// TIA Portal V17 export
// export: Created 2024-06-14T09:52:47.4803756Z, ExportSetting WithDefaults, DisplayName Totally Integrated Automation Portal, DisplayVersion V17, DisplayName TIA Portal Openness, DisplayVersion V17, DisplayName TIA Portal Version Control Interface, DisplayVersion V17, DisplayName Simotion SCOUT TIA, DisplayVersion 5.4.3.0, DisplayName SINAMICS Startdrive Advanced, DisplayVersion V17 SP1 Update 1, DisplayName SINAMICS Startdrive G110M, G120, G120C, G120D, G120P, G115D, DisplayVersion V17 SP1 Update 1, DisplayName SINAMICS Startdrive G130, G150, S120, S150, SINAMICS MV, S210, DisplayVersion V17 SP1 Update 1, DisplayName STEP 7 Professional, DisplayVersion V17, DisplayName STEP 7 Safety, DisplayVersion V17, DisplayName WinCC Professional, DisplayVersion V17
FUNCTION_BLOCK "FILLING_STATION4_FB"   // FB500, LAD
{ S7_Optimized_Access := 'TRUE' }
VERSION : 0.1
// stored: AutoNumber false, IsIECCheckEnabled false, IsRetainMemResEnabled false, MemoryReserve 100, SetENOAutomatically false, UDAEnableTagReadback false
   VAR
      STATION4_S1 { S7_SetPoint := 'True'} : "LPG_FILLING_FB";
      STATION4_S2 { S7_SetPoint := 'True'} : "LPG_FILLING_FB";
      STATION4_S3 { S7_SetPoint := 'True'} : "LPG_FILLING_FB";
      STATION4_S4 { S7_SetPoint := 'True'} : "LPG_FILLING_FB";
      STATION4_S5 { S7_SetPoint := 'True'} : "LPG_FILLING_FB";
      STATION4_S6 { S7_SetPoint := 'True'} : "LPG_FILLING_FB";
      FILLING_STATION4 { S7_SetPoint := 'True'} : "FILLING_FB";
      FILL_SEQ_STARTED { S7_SetPoint := 'True'} : Array[1..6] of Bool;
      FILLING_DONE : Array[1..6] of Bool;
   END_VAR
   VAR_TEMP   // added for the SCL form of the ladder/FBD networks
      _w1 : Bool;
   END_VAR
BEGIN

REGION Network 2: Call Filling Station-4
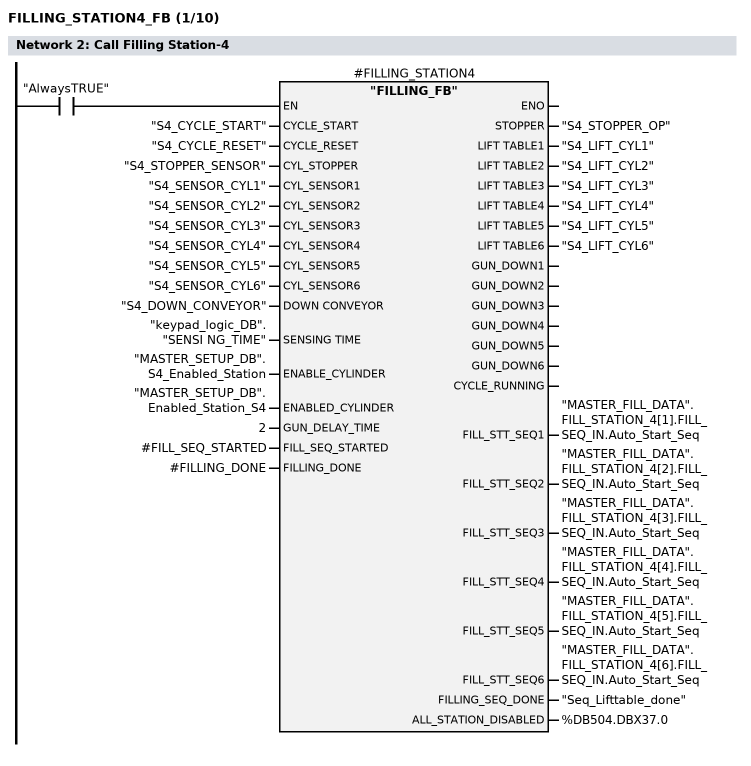
   RUNG wire#powerrail
      Contact( "AlwaysTRUE" )
      #FILLING_STATION4(CYCLE_START := "S4_CYCLE_START", CYCLE_RESET := "S4_CYCLE_RESET", CYL_STOPPER := "S4_STOPPER_SENSOR", CYL_SENSOR1 := "S4_SENSOR_CYL1", CYL_SENSOR2 := "S4_SENSOR_CYL2", CYL_SENSOR3 := "S4_SENSOR_CYL3", CYL_SENSOR4 := "S4_SENSOR_CYL4", CYL_SENSOR5 := "S4_SENSOR_CYL5", CYL_SENSOR6 := "S4_SENSOR_CYL6", "DOWN CONVEYOR" := "S4_DOWN_CONVEYOR", "SENSING TIME" := "keypad_logic_DB"."SENSI NG_TIME", ENABLE_CYLINDER := "MASTER_SETUP_DB".S4_Enabled_Station, ENABLED_CYLINDER := "MASTER_SETUP_DB".Enabled_Station_S4, GUN_DELAY_TIME := 2, FILL_SEQ_STARTED := #FILL_SEQ_STARTED, FILLING_DONE := #FILLING_DONE, STOPPER => "S4_STOPPER_OP", "LIFT TABLE1" => "S4_LIFT_CYL1", "LIFT TABLE2" => "S4_LIFT_CYL2", "LIFT TABLE3" => "S4_LIFT_CYL3", "LIFT TABLE4" => "S4_LIFT_CYL4", "LIFT TABLE5" => "S4_LIFT_CYL5", "LIFT TABLE6" => "S4_LIFT_CYL6", GUN_DOWN1 =>, GUN_DOWN2 =>, GUN_DOWN3 =>, GUN_DOWN4 =>, GUN_DOWN5 =>, GUN_DOWN6 =>, CYCLE_RUNNING =>, FILL_STT_SEQ1 => "MASTER_FILL_DATA".FILL_STATION_4[1].FILL_SEQ_IN.Auto_Start_Seq, FILL_STT_SEQ2 => "MASTER_FILL_DATA".FILL_STATION_4[2].FILL_SEQ_IN.Auto_Start_Seq, FILL_STT_SEQ3 => "MASTER_FILL_DATA".FILL_STATION_4[3].FILL_SEQ_IN.Auto_Start_Seq, FILL_STT_SEQ4 => "MASTER_FILL_DATA".FILL_STATION_4[4].FILL_SEQ_IN.Auto_Start_Seq, FILL_STT_SEQ5 => "MASTER_FILL_DATA".FILL_STATION_4[5].FILL_SEQ_IN.Auto_Start_Seq, FILL_STT_SEQ6 => "MASTER_FILL_DATA".FILL_STATION_4[6].FILL_SEQ_IN.Auto_Start_Seq, FILLING_SEQ_DONE => "Seq_Lifttable_done", ALL_STATION_DISABLED => %DB504.DBX37.0)
   END_RUNG
   // the same network as SCL:
   IF "AlwaysTRUE" THEN
       #FILLING_STATION4(CYCLE_START := "S4_CYCLE_START",   // "FILLING_FB"
                         CYCLE_RESET := "S4_CYCLE_RESET",
                         CYL_STOPPER := "S4_STOPPER_SENSOR",
                         CYL_SENSOR1 := "S4_SENSOR_CYL1",
                         CYL_SENSOR2 := "S4_SENSOR_CYL2",
                         CYL_SENSOR3 := "S4_SENSOR_CYL3",
                         CYL_SENSOR4 := "S4_SENSOR_CYL4",
                         CYL_SENSOR5 := "S4_SENSOR_CYL5",
                         CYL_SENSOR6 := "S4_SENSOR_CYL6",
                         "DOWN CONVEYOR" := "S4_DOWN_CONVEYOR",
                         "SENSING TIME" := "keypad_logic_DB"."SENSI NG_TIME",
                         ENABLE_CYLINDER := "MASTER_SETUP_DB".S4_Enabled_Station,
                         ENABLED_CYLINDER := "MASTER_SETUP_DB".Enabled_Station_S4,
                         GUN_DELAY_TIME := 2,
                         FILL_SEQ_STARTED := #FILL_SEQ_STARTED,
                         FILLING_DONE := #FILLING_DONE,
                         STOPPER => "S4_STOPPER_OP",
                         "LIFT TABLE1" => "S4_LIFT_CYL1",
                         "LIFT TABLE2" => "S4_LIFT_CYL2",
                         "LIFT TABLE3" => "S4_LIFT_CYL3",
                         "LIFT TABLE4" => "S4_LIFT_CYL4",
                         "LIFT TABLE5" => "S4_LIFT_CYL5",
                         "LIFT TABLE6" => "S4_LIFT_CYL6",
                         FILL_STT_SEQ1 => "MASTER_FILL_DATA".FILL_STATION_4[1].FILL_SEQ_IN.Auto_Start_Seq,
                         FILL_STT_SEQ2 => "MASTER_FILL_DATA".FILL_STATION_4[2].FILL_SEQ_IN.Auto_Start_Seq,
                         FILL_STT_SEQ3 => "MASTER_FILL_DATA".FILL_STATION_4[3].FILL_SEQ_IN.Auto_Start_Seq,
                         FILL_STT_SEQ4 => "MASTER_FILL_DATA".FILL_STATION_4[4].FILL_SEQ_IN.Auto_Start_Seq,
                         FILL_STT_SEQ5 => "MASTER_FILL_DATA".FILL_STATION_4[5].FILL_SEQ_IN.Auto_Start_Seq,
                         FILL_STT_SEQ6 => "MASTER_FILL_DATA".FILL_STATION_4[6].FILL_SEQ_IN.Auto_Start_Seq,
                         FILLING_SEQ_DONE => "Seq_Lifttable_done",
                         ALL_STATION_DISABLED => %DB504.DBX37.0);
   END_IF;
END_REGION

REGION Network 3: Call Filling Line-1 Station-1 FB
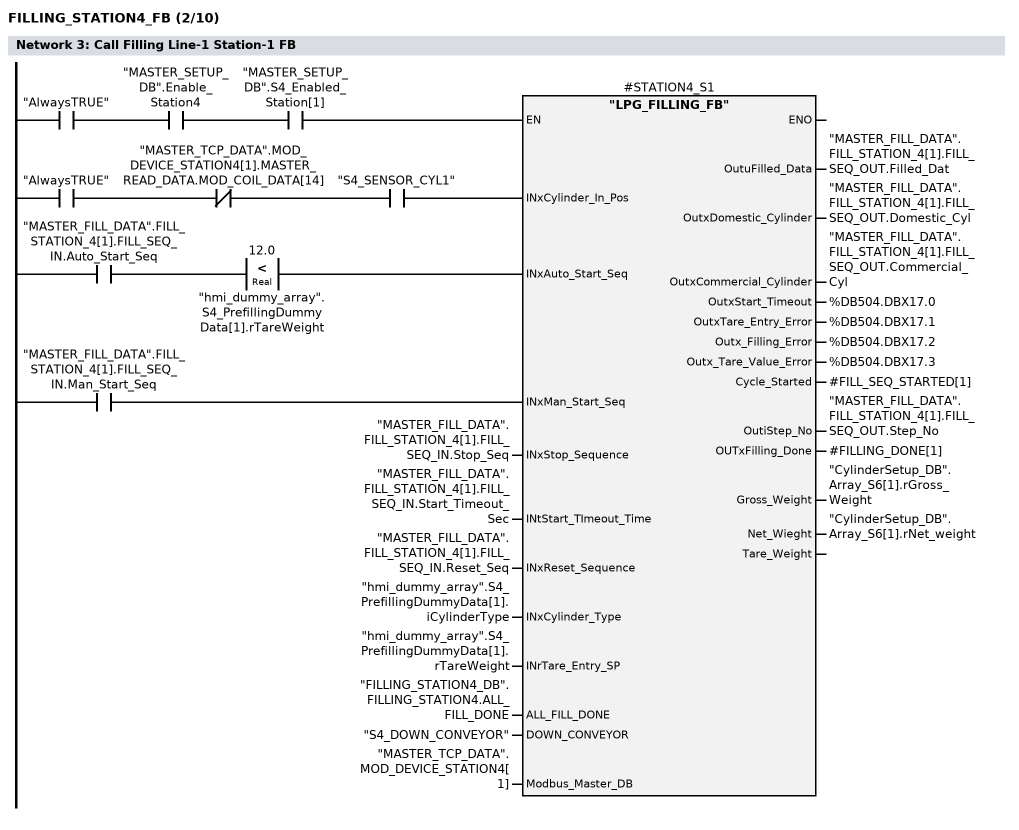
   RUNG wire#powerrail
      Contact( "AlwaysTRUE" )
      Contact( "MASTER_SETUP_DB".Enable_Station4 )
      Contact( "MASTER_SETUP_DB".S4_Enabled_Station[1] )
      #STATION4_S1(INxCylinder_In_Pos := wire#w1, INxAuto_Start_Seq := wire#w2, INxMan_Start_Seq := wire#w3, INxStop_Sequence := "MASTER_FILL_DATA".FILL_STATION_4[1].FILL_SEQ_IN.Stop_Seq, INtStart_TImeout_Time := "MASTER_FILL_DATA".FILL_STATION_4[1].FILL_SEQ_IN.Start_Timeout_Sec, INxReset_Sequence := "MASTER_FILL_DATA".FILL_STATION_4[1].FILL_SEQ_IN.Reset_Seq, INxCylinder_Type := "hmi_dummy_array".S4_PrefillingDummyData[1].iCylinderType, INrTare_Entry_SP := "hmi_dummy_array".S4_PrefillingDummyData[1].rTareWeight, ALL_FILL_DONE := "FILLING_STATION4_DB".FILLING_STATION4.ALL_FILL_DONE, DOWN_CONVEYOR := "S4_DOWN_CONVEYOR", Modbus_Master_DB := "MASTER_TCP_DATA".MOD_DEVICE_STATION4[1], OutuFilled_Data => "MASTER_FILL_DATA".FILL_STATION_4[1].FILL_SEQ_OUT.Filled_Dat, OutxDomestic_Cylinder => "MASTER_FILL_DATA".FILL_STATION_4[1].FILL_SEQ_OUT.Domestic_Cyl, OutxCommercial_Cylinder => "MASTER_FILL_DATA".FILL_STATION_4[1].FILL_SEQ_OUT.Commercial_Cyl, OutxStart_Timeout => %DB504.DBX17.0, OutxTare_Entry_Error => %DB504.DBX17.1, Outx_Filling_Error => %DB504.DBX17.2, Outx_Tare_Value_Error => %DB504.DBX17.3, Cycle_Started => #FILL_SEQ_STARTED[1], OutiStep_No => "MASTER_FILL_DATA".FILL_STATION_4[1].FILL_SEQ_OUT.Step_No, OUTxFilling_Done => #FILLING_DONE[1], Gross_Weight => "CylinderSetup_DB".Array_S6[1].rGross_Weight, Net_Wieght => "CylinderSetup_DB".Array_S6[1].rNet_weight, Tare_Weight =>)
   END_RUNG
   RUNG wire#powerrail
      Contact( "AlwaysTRUE" )
      I_Contact( "MASTER_TCP_DATA".MOD_DEVICE_STATION4[1].MASTER_READ_DATA.MOD_COIL_DATA[14] )
      Contact( "S4_SENSOR_CYL1" )
   END_RUNG wire#w1
   RUNG wire#powerrail
      Contact( "MASTER_FILL_DATA".FILL_STATION_4[1].FILL_SEQ_IN.Auto_Start_Seq )
      { S7_Templates := "SrcType := Real" } LT_Contact(in1 := 12.0, in2 := "hmi_dummy_array".S4_PrefillingDummyData[1].rTareWeight)
   END_RUNG wire#w2
   RUNG wire#powerrail
      Contact( "MASTER_FILL_DATA".FILL_STATION_4[1].FILL_SEQ_IN.Man_Start_Seq )
   END_RUNG wire#w3
   // the same network as SCL:
   IF "AlwaysTRUE" AND "MASTER_SETUP_DB".Enable_Station4 AND "MASTER_SETUP_DB".S4_Enabled_Station[1] THEN
       #STATION4_S1(INxCylinder_In_Pos := "AlwaysTRUE" AND NOT "MASTER_TCP_DATA".MOD_DEVICE_STATION4[1].MASTER_READ_DATA.MOD_COIL_DATA[14] AND "S4_SENSOR_CYL1",   // "LPG_FILLING_FB"
                    INxAuto_Start_Seq := "MASTER_FILL_DATA".FILL_STATION_4[1].FILL_SEQ_IN.Auto_Start_Seq AND (12.0 < "hmi_dummy_array".S4_PrefillingDummyData[1].rTareWeight),
                    INxMan_Start_Seq := "MASTER_FILL_DATA".FILL_STATION_4[1].FILL_SEQ_IN.Man_Start_Seq,
                    INxStop_Sequence := "MASTER_FILL_DATA".FILL_STATION_4[1].FILL_SEQ_IN.Stop_Seq,
                    INtStart_TImeout_Time := "MASTER_FILL_DATA".FILL_STATION_4[1].FILL_SEQ_IN.Start_Timeout_Sec,
                    INxReset_Sequence := "MASTER_FILL_DATA".FILL_STATION_4[1].FILL_SEQ_IN.Reset_Seq,
                    INxCylinder_Type := "hmi_dummy_array".S4_PrefillingDummyData[1].iCylinderType,
                    INrTare_Entry_SP := "hmi_dummy_array".S4_PrefillingDummyData[1].rTareWeight,
                    ALL_FILL_DONE := "FILLING_STATION4_DB".FILLING_STATION4.ALL_FILL_DONE,
                    DOWN_CONVEYOR := "S4_DOWN_CONVEYOR",
                    Modbus_Master_DB := "MASTER_TCP_DATA".MOD_DEVICE_STATION4[1],
                    OutuFilled_Data => "MASTER_FILL_DATA".FILL_STATION_4[1].FILL_SEQ_OUT.Filled_Dat,
                    OutxDomestic_Cylinder => "MASTER_FILL_DATA".FILL_STATION_4[1].FILL_SEQ_OUT.Domestic_Cyl,
                    OutxCommercial_Cylinder => "MASTER_FILL_DATA".FILL_STATION_4[1].FILL_SEQ_OUT.Commercial_Cyl,
                    OutxStart_Timeout => %DB504.DBX17.0,
                    OutxTare_Entry_Error => %DB504.DBX17.1,
                    Outx_Filling_Error => %DB504.DBX17.2,
                    Outx_Tare_Value_Error => %DB504.DBX17.3,
                    Cycle_Started => #FILL_SEQ_STARTED[1],
                    OutiStep_No => "MASTER_FILL_DATA".FILL_STATION_4[1].FILL_SEQ_OUT.Step_No,
                    OUTxFilling_Done => #FILLING_DONE[1],
                    Gross_Weight => "CylinderSetup_DB".Array_S6[1].rGross_Weight,
                    Net_Wieght => "CylinderSetup_DB".Array_S6[1].rNet_weight);
   END_IF;
END_REGION

REGION Network 4: Call Filling Line-1 Station-2 FB
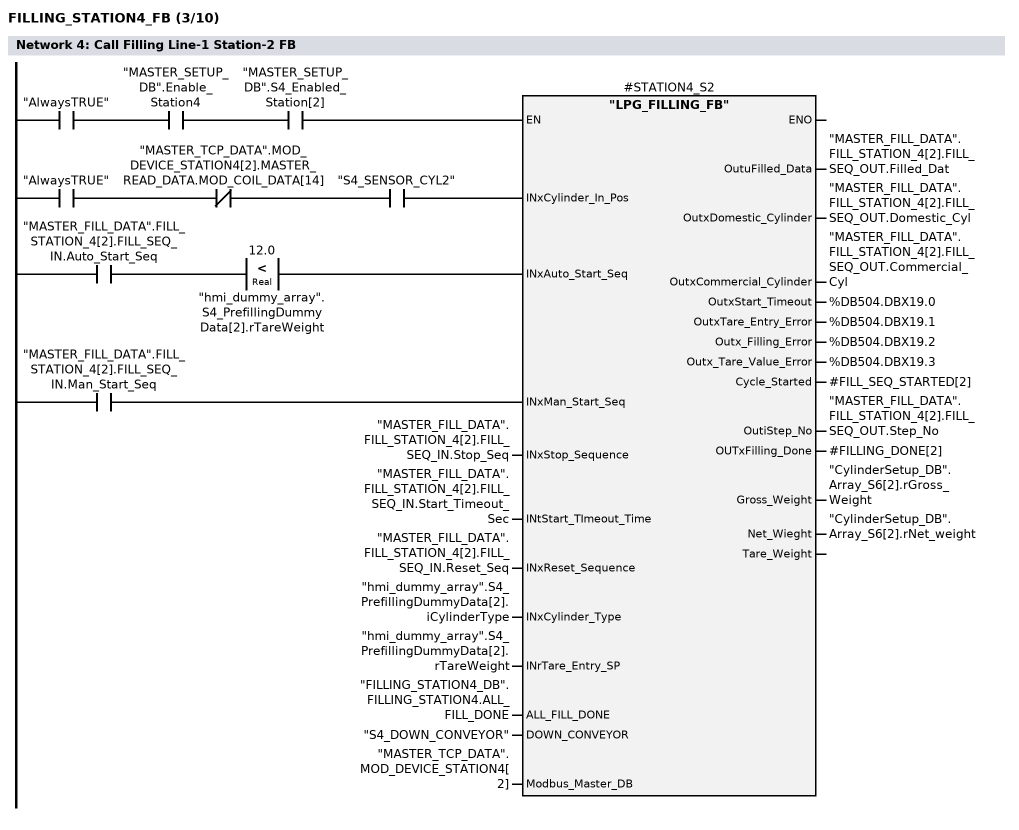
   RUNG wire#powerrail
      Contact( "AlwaysTRUE" )
      Contact( "MASTER_SETUP_DB".Enable_Station4 )
      Contact( "MASTER_SETUP_DB".S4_Enabled_Station[2] )
      #STATION4_S2(INxCylinder_In_Pos := wire#w1, INxAuto_Start_Seq := wire#w2, INxMan_Start_Seq := wire#w3, INxStop_Sequence := "MASTER_FILL_DATA".FILL_STATION_4[2].FILL_SEQ_IN.Stop_Seq, INtStart_TImeout_Time := "MASTER_FILL_DATA".FILL_STATION_4[2].FILL_SEQ_IN.Start_Timeout_Sec, INxReset_Sequence := "MASTER_FILL_DATA".FILL_STATION_4[2].FILL_SEQ_IN.Reset_Seq, INxCylinder_Type := "hmi_dummy_array".S4_PrefillingDummyData[2].iCylinderType, INrTare_Entry_SP := "hmi_dummy_array".S4_PrefillingDummyData[2].rTareWeight, ALL_FILL_DONE := "FILLING_STATION4_DB".FILLING_STATION4.ALL_FILL_DONE, DOWN_CONVEYOR := "S4_DOWN_CONVEYOR", Modbus_Master_DB := "MASTER_TCP_DATA".MOD_DEVICE_STATION4[2], OutuFilled_Data => "MASTER_FILL_DATA".FILL_STATION_4[2].FILL_SEQ_OUT.Filled_Dat, OutxDomestic_Cylinder => "MASTER_FILL_DATA".FILL_STATION_4[2].FILL_SEQ_OUT.Domestic_Cyl, OutxCommercial_Cylinder => "MASTER_FILL_DATA".FILL_STATION_4[2].FILL_SEQ_OUT.Commercial_Cyl, OutxStart_Timeout => %DB504.DBX19.0, OutxTare_Entry_Error => %DB504.DBX19.1, Outx_Filling_Error => %DB504.DBX19.2, Outx_Tare_Value_Error => %DB504.DBX19.3, Cycle_Started => #FILL_SEQ_STARTED[2], OutiStep_No => "MASTER_FILL_DATA".FILL_STATION_4[2].FILL_SEQ_OUT.Step_No, OUTxFilling_Done => #FILLING_DONE[2], Gross_Weight => "CylinderSetup_DB".Array_S6[2].rGross_Weight, Net_Wieght => "CylinderSetup_DB".Array_S6[2].rNet_weight, Tare_Weight =>)
   END_RUNG
   RUNG wire#powerrail
      Contact( "AlwaysTRUE" )
      I_Contact( "MASTER_TCP_DATA".MOD_DEVICE_STATION4[2].MASTER_READ_DATA.MOD_COIL_DATA[14] )
      Contact( "S4_SENSOR_CYL2" )
   END_RUNG wire#w1
   RUNG wire#powerrail
      Contact( "MASTER_FILL_DATA".FILL_STATION_4[2].FILL_SEQ_IN.Auto_Start_Seq )
      { S7_Templates := "SrcType := Real" } LT_Contact(in1 := 12.0, in2 := "hmi_dummy_array".S4_PrefillingDummyData[2].rTareWeight)
   END_RUNG wire#w2
   RUNG wire#powerrail
      Contact( "MASTER_FILL_DATA".FILL_STATION_4[2].FILL_SEQ_IN.Man_Start_Seq )
   END_RUNG wire#w3
   // the same network as SCL:
   IF "AlwaysTRUE" AND "MASTER_SETUP_DB".Enable_Station4 AND "MASTER_SETUP_DB".S4_Enabled_Station[2] THEN
       #STATION4_S2(INxCylinder_In_Pos := "AlwaysTRUE" AND NOT "MASTER_TCP_DATA".MOD_DEVICE_STATION4[2].MASTER_READ_DATA.MOD_COIL_DATA[14] AND "S4_SENSOR_CYL2",   // "LPG_FILLING_FB"
                    INxAuto_Start_Seq := "MASTER_FILL_DATA".FILL_STATION_4[2].FILL_SEQ_IN.Auto_Start_Seq AND (12.0 < "hmi_dummy_array".S4_PrefillingDummyData[2].rTareWeight),
                    INxMan_Start_Seq := "MASTER_FILL_DATA".FILL_STATION_4[2].FILL_SEQ_IN.Man_Start_Seq,
                    INxStop_Sequence := "MASTER_FILL_DATA".FILL_STATION_4[2].FILL_SEQ_IN.Stop_Seq,
                    INtStart_TImeout_Time := "MASTER_FILL_DATA".FILL_STATION_4[2].FILL_SEQ_IN.Start_Timeout_Sec,
                    INxReset_Sequence := "MASTER_FILL_DATA".FILL_STATION_4[2].FILL_SEQ_IN.Reset_Seq,
                    INxCylinder_Type := "hmi_dummy_array".S4_PrefillingDummyData[2].iCylinderType,
                    INrTare_Entry_SP := "hmi_dummy_array".S4_PrefillingDummyData[2].rTareWeight,
                    ALL_FILL_DONE := "FILLING_STATION4_DB".FILLING_STATION4.ALL_FILL_DONE,
                    DOWN_CONVEYOR := "S4_DOWN_CONVEYOR",
                    Modbus_Master_DB := "MASTER_TCP_DATA".MOD_DEVICE_STATION4[2],
                    OutuFilled_Data => "MASTER_FILL_DATA".FILL_STATION_4[2].FILL_SEQ_OUT.Filled_Dat,
                    OutxDomestic_Cylinder => "MASTER_FILL_DATA".FILL_STATION_4[2].FILL_SEQ_OUT.Domestic_Cyl,
                    OutxCommercial_Cylinder => "MASTER_FILL_DATA".FILL_STATION_4[2].FILL_SEQ_OUT.Commercial_Cyl,
                    OutxStart_Timeout => %DB504.DBX19.0,
                    OutxTare_Entry_Error => %DB504.DBX19.1,
                    Outx_Filling_Error => %DB504.DBX19.2,
                    Outx_Tare_Value_Error => %DB504.DBX19.3,
                    Cycle_Started => #FILL_SEQ_STARTED[2],
                    OutiStep_No => "MASTER_FILL_DATA".FILL_STATION_4[2].FILL_SEQ_OUT.Step_No,
                    OUTxFilling_Done => #FILLING_DONE[2],
                    Gross_Weight => "CylinderSetup_DB".Array_S6[2].rGross_Weight,
                    Net_Wieght => "CylinderSetup_DB".Array_S6[2].rNet_weight);
   END_IF;
END_REGION

REGION Network 5: Call Filling Line-1 Station-3 FB
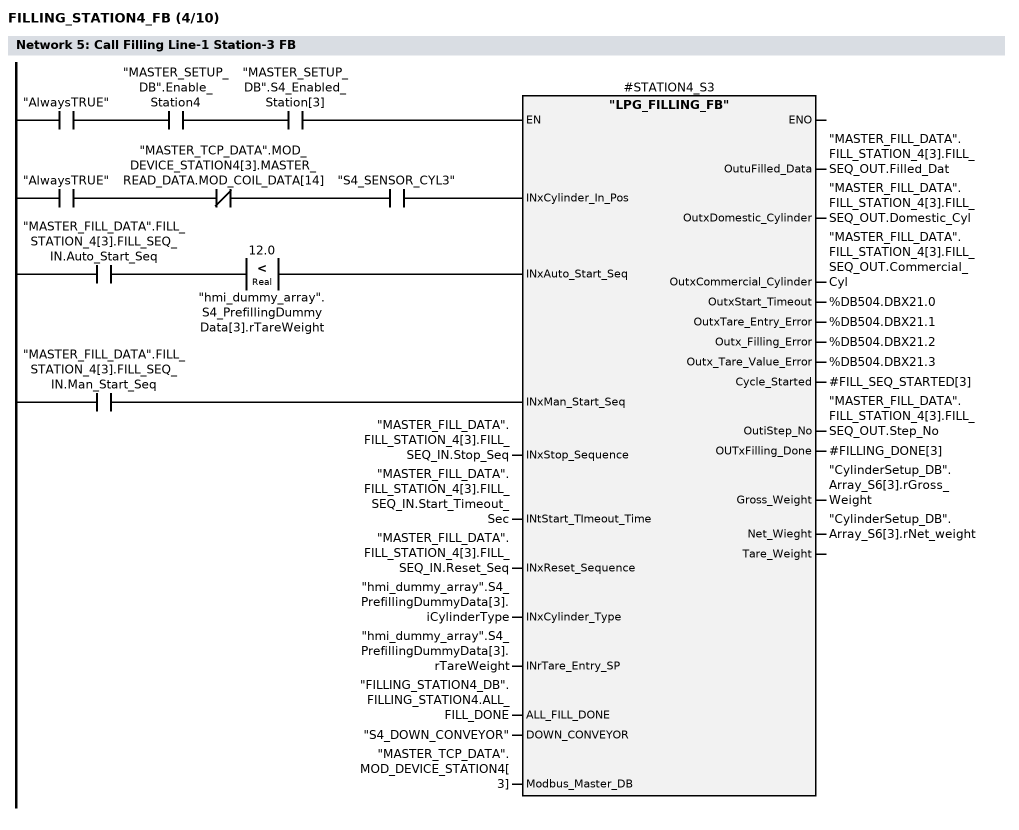
   RUNG wire#powerrail
      Contact( "AlwaysTRUE" )
      Contact( "MASTER_SETUP_DB".Enable_Station4 )
      Contact( "MASTER_SETUP_DB".S4_Enabled_Station[3] )
      #STATION4_S3(INxCylinder_In_Pos := wire#w1, INxAuto_Start_Seq := wire#w2, INxMan_Start_Seq := wire#w3, INxStop_Sequence := "MASTER_FILL_DATA".FILL_STATION_4[3].FILL_SEQ_IN.Stop_Seq, INtStart_TImeout_Time := "MASTER_FILL_DATA".FILL_STATION_4[3].FILL_SEQ_IN.Start_Timeout_Sec, INxReset_Sequence := "MASTER_FILL_DATA".FILL_STATION_4[3].FILL_SEQ_IN.Reset_Seq, INxCylinder_Type := "hmi_dummy_array".S4_PrefillingDummyData[3].iCylinderType, INrTare_Entry_SP := "hmi_dummy_array".S4_PrefillingDummyData[3].rTareWeight, ALL_FILL_DONE := "FILLING_STATION4_DB".FILLING_STATION4.ALL_FILL_DONE, DOWN_CONVEYOR := "S4_DOWN_CONVEYOR", Modbus_Master_DB := "MASTER_TCP_DATA".MOD_DEVICE_STATION4[3], OutuFilled_Data => "MASTER_FILL_DATA".FILL_STATION_4[3].FILL_SEQ_OUT.Filled_Dat, OutxDomestic_Cylinder => "MASTER_FILL_DATA".FILL_STATION_4[3].FILL_SEQ_OUT.Domestic_Cyl, OutxCommercial_Cylinder => "MASTER_FILL_DATA".FILL_STATION_4[3].FILL_SEQ_OUT.Commercial_Cyl, OutxStart_Timeout => %DB504.DBX21.0, OutxTare_Entry_Error => %DB504.DBX21.1, Outx_Filling_Error => %DB504.DBX21.2, Outx_Tare_Value_Error => %DB504.DBX21.3, Cycle_Started => #FILL_SEQ_STARTED[3], OutiStep_No => "MASTER_FILL_DATA".FILL_STATION_4[3].FILL_SEQ_OUT.Step_No, OUTxFilling_Done => #FILLING_DONE[3], Gross_Weight => "CylinderSetup_DB".Array_S6[3].rGross_Weight, Net_Wieght => "CylinderSetup_DB".Array_S6[3].rNet_weight, Tare_Weight =>)
   END_RUNG
   RUNG wire#powerrail
      Contact( "AlwaysTRUE" )
      I_Contact( "MASTER_TCP_DATA".MOD_DEVICE_STATION4[3].MASTER_READ_DATA.MOD_COIL_DATA[14] )
      Contact( "S4_SENSOR_CYL3" )
   END_RUNG wire#w1
   RUNG wire#powerrail
      Contact( "MASTER_FILL_DATA".FILL_STATION_4[3].FILL_SEQ_IN.Auto_Start_Seq )
      { S7_Templates := "SrcType := Real" } LT_Contact(in1 := 12.0, in2 := "hmi_dummy_array".S4_PrefillingDummyData[3].rTareWeight)
   END_RUNG wire#w2
   RUNG wire#powerrail
      Contact( "MASTER_FILL_DATA".FILL_STATION_4[3].FILL_SEQ_IN.Man_Start_Seq )
   END_RUNG wire#w3
   // the same network as SCL:
   IF "AlwaysTRUE" AND "MASTER_SETUP_DB".Enable_Station4 AND "MASTER_SETUP_DB".S4_Enabled_Station[3] THEN
       #STATION4_S3(INxCylinder_In_Pos := "AlwaysTRUE" AND NOT "MASTER_TCP_DATA".MOD_DEVICE_STATION4[3].MASTER_READ_DATA.MOD_COIL_DATA[14] AND "S4_SENSOR_CYL3",   // "LPG_FILLING_FB"
                    INxAuto_Start_Seq := "MASTER_FILL_DATA".FILL_STATION_4[3].FILL_SEQ_IN.Auto_Start_Seq AND (12.0 < "hmi_dummy_array".S4_PrefillingDummyData[3].rTareWeight),
                    INxMan_Start_Seq := "MASTER_FILL_DATA".FILL_STATION_4[3].FILL_SEQ_IN.Man_Start_Seq,
                    INxStop_Sequence := "MASTER_FILL_DATA".FILL_STATION_4[3].FILL_SEQ_IN.Stop_Seq,
                    INtStart_TImeout_Time := "MASTER_FILL_DATA".FILL_STATION_4[3].FILL_SEQ_IN.Start_Timeout_Sec,
                    INxReset_Sequence := "MASTER_FILL_DATA".FILL_STATION_4[3].FILL_SEQ_IN.Reset_Seq,
                    INxCylinder_Type := "hmi_dummy_array".S4_PrefillingDummyData[3].iCylinderType,
                    INrTare_Entry_SP := "hmi_dummy_array".S4_PrefillingDummyData[3].rTareWeight,
                    ALL_FILL_DONE := "FILLING_STATION4_DB".FILLING_STATION4.ALL_FILL_DONE,
                    DOWN_CONVEYOR := "S4_DOWN_CONVEYOR",
                    Modbus_Master_DB := "MASTER_TCP_DATA".MOD_DEVICE_STATION4[3],
                    OutuFilled_Data => "MASTER_FILL_DATA".FILL_STATION_4[3].FILL_SEQ_OUT.Filled_Dat,
                    OutxDomestic_Cylinder => "MASTER_FILL_DATA".FILL_STATION_4[3].FILL_SEQ_OUT.Domestic_Cyl,
                    OutxCommercial_Cylinder => "MASTER_FILL_DATA".FILL_STATION_4[3].FILL_SEQ_OUT.Commercial_Cyl,
                    OutxStart_Timeout => %DB504.DBX21.0,
                    OutxTare_Entry_Error => %DB504.DBX21.1,
                    Outx_Filling_Error => %DB504.DBX21.2,
                    Outx_Tare_Value_Error => %DB504.DBX21.3,
                    Cycle_Started => #FILL_SEQ_STARTED[3],
                    OutiStep_No => "MASTER_FILL_DATA".FILL_STATION_4[3].FILL_SEQ_OUT.Step_No,
                    OUTxFilling_Done => #FILLING_DONE[3],
                    Gross_Weight => "CylinderSetup_DB".Array_S6[3].rGross_Weight,
                    Net_Wieght => "CylinderSetup_DB".Array_S6[3].rNet_weight);
   END_IF;
END_REGION

REGION Network 6: Call Filling Line-1 Station-4 FB
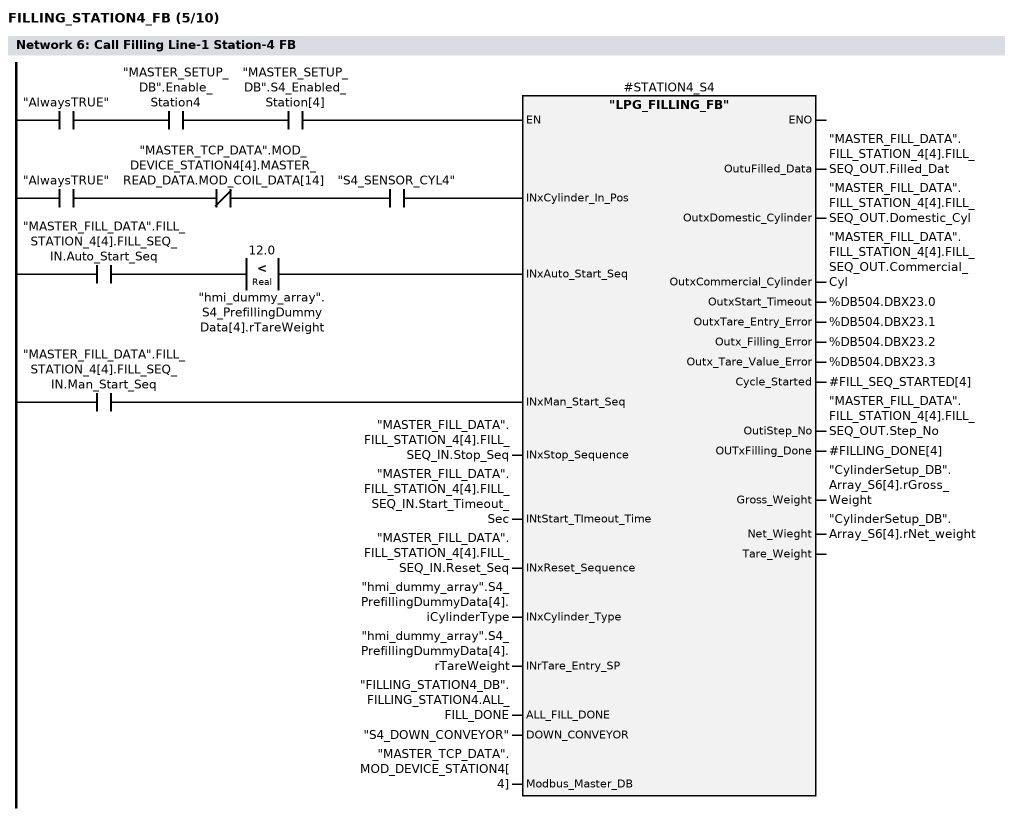
   RUNG wire#powerrail
      Contact( "AlwaysTRUE" )
      Contact( "MASTER_SETUP_DB".Enable_Station4 )
      Contact( "MASTER_SETUP_DB".S4_Enabled_Station[4] )
      #STATION4_S4(INxCylinder_In_Pos := wire#w1, INxAuto_Start_Seq := wire#w2, INxMan_Start_Seq := wire#w3, INxStop_Sequence := "MASTER_FILL_DATA".FILL_STATION_4[4].FILL_SEQ_IN.Stop_Seq, INtStart_TImeout_Time := "MASTER_FILL_DATA".FILL_STATION_4[4].FILL_SEQ_IN.Start_Timeout_Sec, INxReset_Sequence := "MASTER_FILL_DATA".FILL_STATION_4[4].FILL_SEQ_IN.Reset_Seq, INxCylinder_Type := "hmi_dummy_array".S4_PrefillingDummyData[4].iCylinderType, INrTare_Entry_SP := "hmi_dummy_array".S4_PrefillingDummyData[4].rTareWeight, ALL_FILL_DONE := "FILLING_STATION4_DB".FILLING_STATION4.ALL_FILL_DONE, DOWN_CONVEYOR := "S4_DOWN_CONVEYOR", Modbus_Master_DB := "MASTER_TCP_DATA".MOD_DEVICE_STATION4[4], OutuFilled_Data => "MASTER_FILL_DATA".FILL_STATION_4[4].FILL_SEQ_OUT.Filled_Dat, OutxDomestic_Cylinder => "MASTER_FILL_DATA".FILL_STATION_4[4].FILL_SEQ_OUT.Domestic_Cyl, OutxCommercial_Cylinder => "MASTER_FILL_DATA".FILL_STATION_4[4].FILL_SEQ_OUT.Commercial_Cyl, OutxStart_Timeout => %DB504.DBX23.0, OutxTare_Entry_Error => %DB504.DBX23.1, Outx_Filling_Error => %DB504.DBX23.2, Outx_Tare_Value_Error => %DB504.DBX23.3, Cycle_Started => #FILL_SEQ_STARTED[4], OutiStep_No => "MASTER_FILL_DATA".FILL_STATION_4[4].FILL_SEQ_OUT.Step_No, OUTxFilling_Done => #FILLING_DONE[4], Gross_Weight => "CylinderSetup_DB".Array_S6[4].rGross_Weight, Net_Wieght => "CylinderSetup_DB".Array_S6[4].rNet_weight, Tare_Weight =>)
   END_RUNG
   RUNG wire#powerrail
      Contact( "AlwaysTRUE" )
      I_Contact( "MASTER_TCP_DATA".MOD_DEVICE_STATION4[4].MASTER_READ_DATA.MOD_COIL_DATA[14] )
      Contact( "S4_SENSOR_CYL4" )
   END_RUNG wire#w1
   RUNG wire#powerrail
      Contact( "MASTER_FILL_DATA".FILL_STATION_4[4].FILL_SEQ_IN.Auto_Start_Seq )
      { S7_Templates := "SrcType := Real" } LT_Contact(in1 := 12.0, in2 := "hmi_dummy_array".S4_PrefillingDummyData[4].rTareWeight)
   END_RUNG wire#w2
   RUNG wire#powerrail
      Contact( "MASTER_FILL_DATA".FILL_STATION_4[4].FILL_SEQ_IN.Man_Start_Seq )
   END_RUNG wire#w3
   // the same network as SCL:
   IF "AlwaysTRUE" AND "MASTER_SETUP_DB".Enable_Station4 AND "MASTER_SETUP_DB".S4_Enabled_Station[4] THEN
       #STATION4_S4(INxCylinder_In_Pos := "AlwaysTRUE" AND NOT "MASTER_TCP_DATA".MOD_DEVICE_STATION4[4].MASTER_READ_DATA.MOD_COIL_DATA[14] AND "S4_SENSOR_CYL4",   // "LPG_FILLING_FB"
                    INxAuto_Start_Seq := "MASTER_FILL_DATA".FILL_STATION_4[4].FILL_SEQ_IN.Auto_Start_Seq AND (12.0 < "hmi_dummy_array".S4_PrefillingDummyData[4].rTareWeight),
                    INxMan_Start_Seq := "MASTER_FILL_DATA".FILL_STATION_4[4].FILL_SEQ_IN.Man_Start_Seq,
                    INxStop_Sequence := "MASTER_FILL_DATA".FILL_STATION_4[4].FILL_SEQ_IN.Stop_Seq,
                    INtStart_TImeout_Time := "MASTER_FILL_DATA".FILL_STATION_4[4].FILL_SEQ_IN.Start_Timeout_Sec,
                    INxReset_Sequence := "MASTER_FILL_DATA".FILL_STATION_4[4].FILL_SEQ_IN.Reset_Seq,
                    INxCylinder_Type := "hmi_dummy_array".S4_PrefillingDummyData[4].iCylinderType,
                    INrTare_Entry_SP := "hmi_dummy_array".S4_PrefillingDummyData[4].rTareWeight,
                    ALL_FILL_DONE := "FILLING_STATION4_DB".FILLING_STATION4.ALL_FILL_DONE,
                    DOWN_CONVEYOR := "S4_DOWN_CONVEYOR",
                    Modbus_Master_DB := "MASTER_TCP_DATA".MOD_DEVICE_STATION4[4],
                    OutuFilled_Data => "MASTER_FILL_DATA".FILL_STATION_4[4].FILL_SEQ_OUT.Filled_Dat,
                    OutxDomestic_Cylinder => "MASTER_FILL_DATA".FILL_STATION_4[4].FILL_SEQ_OUT.Domestic_Cyl,
                    OutxCommercial_Cylinder => "MASTER_FILL_DATA".FILL_STATION_4[4].FILL_SEQ_OUT.Commercial_Cyl,
                    OutxStart_Timeout => %DB504.DBX23.0,
                    OutxTare_Entry_Error => %DB504.DBX23.1,
                    Outx_Filling_Error => %DB504.DBX23.2,
                    Outx_Tare_Value_Error => %DB504.DBX23.3,
                    Cycle_Started => #FILL_SEQ_STARTED[4],
                    OutiStep_No => "MASTER_FILL_DATA".FILL_STATION_4[4].FILL_SEQ_OUT.Step_No,
                    OUTxFilling_Done => #FILLING_DONE[4],
                    Gross_Weight => "CylinderSetup_DB".Array_S6[4].rGross_Weight,
                    Net_Wieght => "CylinderSetup_DB".Array_S6[4].rNet_weight);
   END_IF;
END_REGION

REGION Network 7: Call Filling Line-1 Station-5 FB
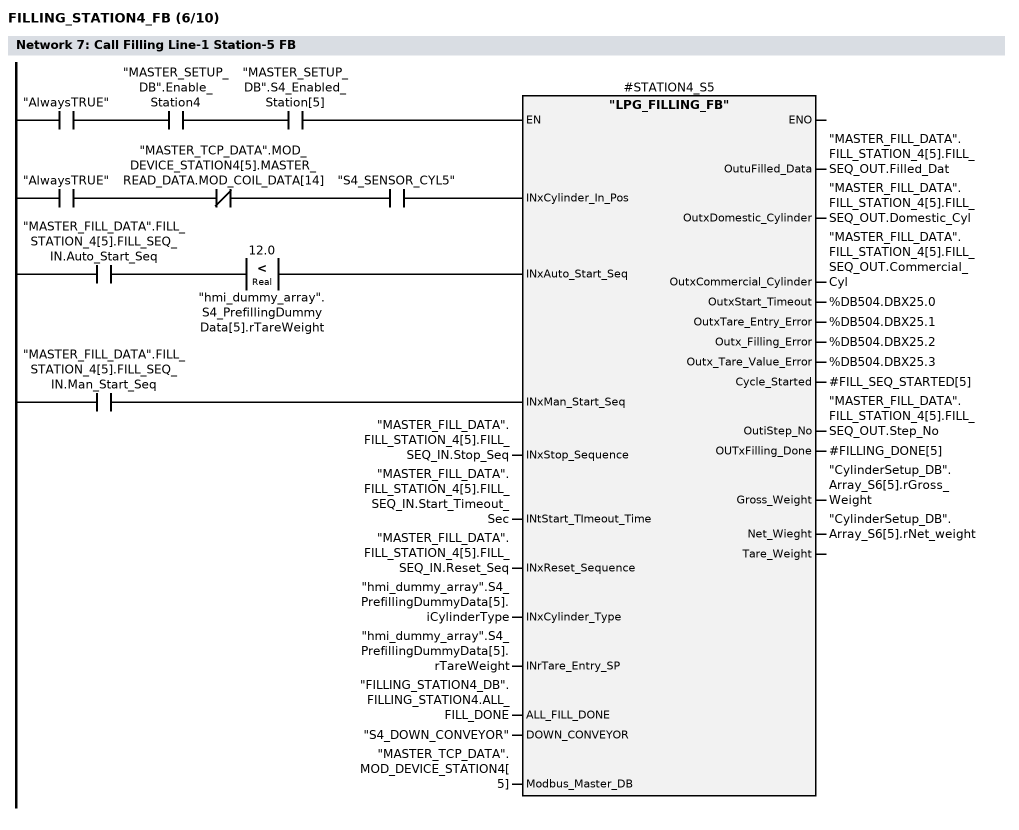
   RUNG wire#powerrail
      Contact( "AlwaysTRUE" )
      Contact( "MASTER_SETUP_DB".Enable_Station4 )
      Contact( "MASTER_SETUP_DB".S4_Enabled_Station[5] )
      #STATION4_S5(INxCylinder_In_Pos := wire#w1, INxAuto_Start_Seq := wire#w2, INxMan_Start_Seq := wire#w3, INxStop_Sequence := "MASTER_FILL_DATA".FILL_STATION_4[5].FILL_SEQ_IN.Stop_Seq, INtStart_TImeout_Time := "MASTER_FILL_DATA".FILL_STATION_4[5].FILL_SEQ_IN.Start_Timeout_Sec, INxReset_Sequence := "MASTER_FILL_DATA".FILL_STATION_4[5].FILL_SEQ_IN.Reset_Seq, INxCylinder_Type := "hmi_dummy_array".S4_PrefillingDummyData[5].iCylinderType, INrTare_Entry_SP := "hmi_dummy_array".S4_PrefillingDummyData[5].rTareWeight, ALL_FILL_DONE := "FILLING_STATION4_DB".FILLING_STATION4.ALL_FILL_DONE, DOWN_CONVEYOR := "S4_DOWN_CONVEYOR", Modbus_Master_DB := "MASTER_TCP_DATA".MOD_DEVICE_STATION4[5], OutuFilled_Data => "MASTER_FILL_DATA".FILL_STATION_4[5].FILL_SEQ_OUT.Filled_Dat, OutxDomestic_Cylinder => "MASTER_FILL_DATA".FILL_STATION_4[5].FILL_SEQ_OUT.Domestic_Cyl, OutxCommercial_Cylinder => "MASTER_FILL_DATA".FILL_STATION_4[5].FILL_SEQ_OUT.Commercial_Cyl, OutxStart_Timeout => %DB504.DBX25.0, OutxTare_Entry_Error => %DB504.DBX25.1, Outx_Filling_Error => %DB504.DBX25.2, Outx_Tare_Value_Error => %DB504.DBX25.3, Cycle_Started => #FILL_SEQ_STARTED[5], OutiStep_No => "MASTER_FILL_DATA".FILL_STATION_4[5].FILL_SEQ_OUT.Step_No, OUTxFilling_Done => #FILLING_DONE[5], Gross_Weight => "CylinderSetup_DB".Array_S6[5].rGross_Weight, Net_Wieght => "CylinderSetup_DB".Array_S6[5].rNet_weight, Tare_Weight =>)
   END_RUNG
   RUNG wire#powerrail
      Contact( "AlwaysTRUE" )
      I_Contact( "MASTER_TCP_DATA".MOD_DEVICE_STATION4[5].MASTER_READ_DATA.MOD_COIL_DATA[14] )
      Contact( "S4_SENSOR_CYL5" )
   END_RUNG wire#w1
   RUNG wire#powerrail
      Contact( "MASTER_FILL_DATA".FILL_STATION_4[5].FILL_SEQ_IN.Auto_Start_Seq )
      { S7_Templates := "SrcType := Real" } LT_Contact(in1 := 12.0, in2 := "hmi_dummy_array".S4_PrefillingDummyData[5].rTareWeight)
   END_RUNG wire#w2
   RUNG wire#powerrail
      Contact( "MASTER_FILL_DATA".FILL_STATION_4[5].FILL_SEQ_IN.Man_Start_Seq )
   END_RUNG wire#w3
   // the same network as SCL:
   IF "AlwaysTRUE" AND "MASTER_SETUP_DB".Enable_Station4 AND "MASTER_SETUP_DB".S4_Enabled_Station[5] THEN
       #STATION4_S5(INxCylinder_In_Pos := "AlwaysTRUE" AND NOT "MASTER_TCP_DATA".MOD_DEVICE_STATION4[5].MASTER_READ_DATA.MOD_COIL_DATA[14] AND "S4_SENSOR_CYL5",   // "LPG_FILLING_FB"
                    INxAuto_Start_Seq := "MASTER_FILL_DATA".FILL_STATION_4[5].FILL_SEQ_IN.Auto_Start_Seq AND (12.0 < "hmi_dummy_array".S4_PrefillingDummyData[5].rTareWeight),
                    INxMan_Start_Seq := "MASTER_FILL_DATA".FILL_STATION_4[5].FILL_SEQ_IN.Man_Start_Seq,
                    INxStop_Sequence := "MASTER_FILL_DATA".FILL_STATION_4[5].FILL_SEQ_IN.Stop_Seq,
                    INtStart_TImeout_Time := "MASTER_FILL_DATA".FILL_STATION_4[5].FILL_SEQ_IN.Start_Timeout_Sec,
                    INxReset_Sequence := "MASTER_FILL_DATA".FILL_STATION_4[5].FILL_SEQ_IN.Reset_Seq,
                    INxCylinder_Type := "hmi_dummy_array".S4_PrefillingDummyData[5].iCylinderType,
                    INrTare_Entry_SP := "hmi_dummy_array".S4_PrefillingDummyData[5].rTareWeight,
                    ALL_FILL_DONE := "FILLING_STATION4_DB".FILLING_STATION4.ALL_FILL_DONE,
                    DOWN_CONVEYOR := "S4_DOWN_CONVEYOR",
                    Modbus_Master_DB := "MASTER_TCP_DATA".MOD_DEVICE_STATION4[5],
                    OutuFilled_Data => "MASTER_FILL_DATA".FILL_STATION_4[5].FILL_SEQ_OUT.Filled_Dat,
                    OutxDomestic_Cylinder => "MASTER_FILL_DATA".FILL_STATION_4[5].FILL_SEQ_OUT.Domestic_Cyl,
                    OutxCommercial_Cylinder => "MASTER_FILL_DATA".FILL_STATION_4[5].FILL_SEQ_OUT.Commercial_Cyl,
                    OutxStart_Timeout => %DB504.DBX25.0,
                    OutxTare_Entry_Error => %DB504.DBX25.1,
                    Outx_Filling_Error => %DB504.DBX25.2,
                    Outx_Tare_Value_Error => %DB504.DBX25.3,
                    Cycle_Started => #FILL_SEQ_STARTED[5],
                    OutiStep_No => "MASTER_FILL_DATA".FILL_STATION_4[5].FILL_SEQ_OUT.Step_No,
                    OUTxFilling_Done => #FILLING_DONE[5],
                    Gross_Weight => "CylinderSetup_DB".Array_S6[5].rGross_Weight,
                    Net_Wieght => "CylinderSetup_DB".Array_S6[5].rNet_weight);
   END_IF;
END_REGION

REGION Network 8: Call Filling Line-1 Station-6 FB
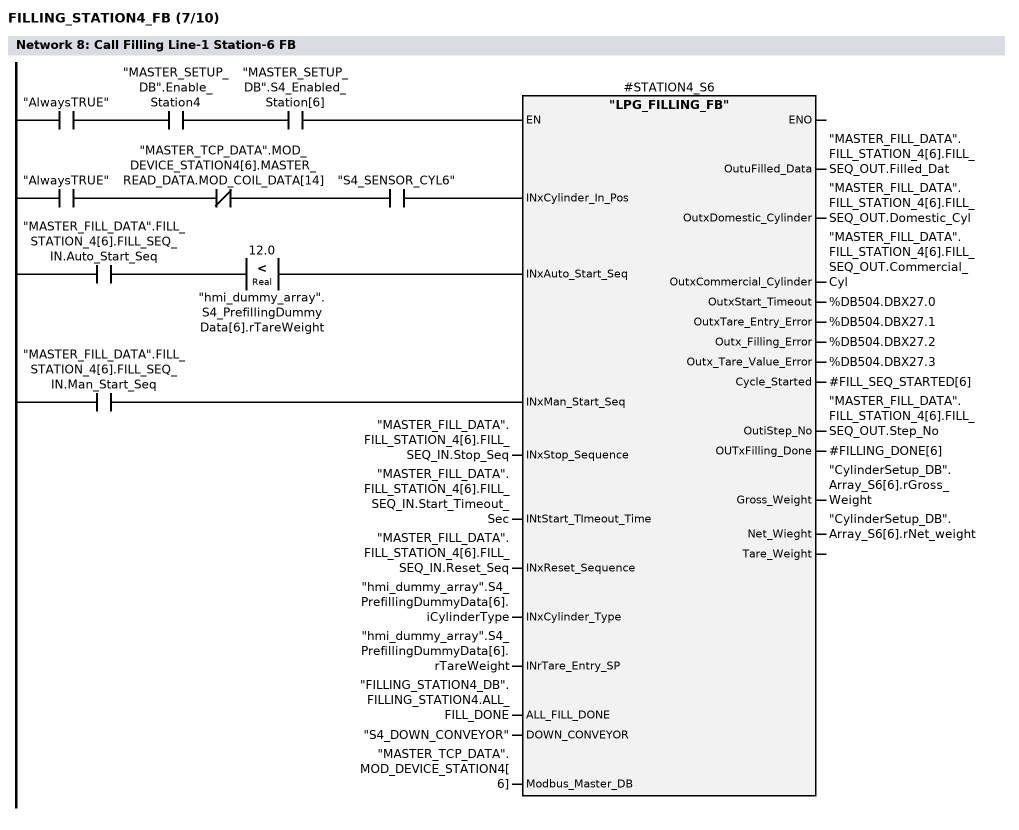
   RUNG wire#powerrail
      Contact( "AlwaysTRUE" )
      Contact( "MASTER_SETUP_DB".Enable_Station4 )
      Contact( "MASTER_SETUP_DB".S4_Enabled_Station[6] )
      #STATION4_S6(INxCylinder_In_Pos := wire#w1, INxAuto_Start_Seq := wire#w2, INxMan_Start_Seq := wire#w3, INxStop_Sequence := "MASTER_FILL_DATA".FILL_STATION_4[6].FILL_SEQ_IN.Stop_Seq, INtStart_TImeout_Time := "MASTER_FILL_DATA".FILL_STATION_4[6].FILL_SEQ_IN.Start_Timeout_Sec, INxReset_Sequence := "MASTER_FILL_DATA".FILL_STATION_4[6].FILL_SEQ_IN.Reset_Seq, INxCylinder_Type := "hmi_dummy_array".S4_PrefillingDummyData[6].iCylinderType, INrTare_Entry_SP := "hmi_dummy_array".S4_PrefillingDummyData[6].rTareWeight, ALL_FILL_DONE := "FILLING_STATION4_DB".FILLING_STATION4.ALL_FILL_DONE, DOWN_CONVEYOR := "S4_DOWN_CONVEYOR", Modbus_Master_DB := "MASTER_TCP_DATA".MOD_DEVICE_STATION4[6], OutuFilled_Data => "MASTER_FILL_DATA".FILL_STATION_4[6].FILL_SEQ_OUT.Filled_Dat, OutxDomestic_Cylinder => "MASTER_FILL_DATA".FILL_STATION_4[6].FILL_SEQ_OUT.Domestic_Cyl, OutxCommercial_Cylinder => "MASTER_FILL_DATA".FILL_STATION_4[6].FILL_SEQ_OUT.Commercial_Cyl, OutxStart_Timeout => %DB504.DBX27.0, OutxTare_Entry_Error => %DB504.DBX27.1, Outx_Filling_Error => %DB504.DBX27.2, Outx_Tare_Value_Error => %DB504.DBX27.3, Cycle_Started => #FILL_SEQ_STARTED[6], OutiStep_No => "MASTER_FILL_DATA".FILL_STATION_4[6].FILL_SEQ_OUT.Step_No, OUTxFilling_Done => #FILLING_DONE[6], Gross_Weight => "CylinderSetup_DB".Array_S6[6].rGross_Weight, Net_Wieght => "CylinderSetup_DB".Array_S6[6].rNet_weight, Tare_Weight =>)
   END_RUNG
   RUNG wire#powerrail
      Contact( "AlwaysTRUE" )
      I_Contact( "MASTER_TCP_DATA".MOD_DEVICE_STATION4[6].MASTER_READ_DATA.MOD_COIL_DATA[14] )
      Contact( "S4_SENSOR_CYL6" )
   END_RUNG wire#w1
   RUNG wire#powerrail
      Contact( "MASTER_FILL_DATA".FILL_STATION_4[6].FILL_SEQ_IN.Auto_Start_Seq )
      { S7_Templates := "SrcType := Real" } LT_Contact(in1 := 12.0, in2 := "hmi_dummy_array".S4_PrefillingDummyData[6].rTareWeight)
   END_RUNG wire#w2
   RUNG wire#powerrail
      Contact( "MASTER_FILL_DATA".FILL_STATION_4[6].FILL_SEQ_IN.Man_Start_Seq )
   END_RUNG wire#w3
   // the same network as SCL:
   IF "AlwaysTRUE" AND "MASTER_SETUP_DB".Enable_Station4 AND "MASTER_SETUP_DB".S4_Enabled_Station[6] THEN
       #STATION4_S6(INxCylinder_In_Pos := "AlwaysTRUE" AND NOT "MASTER_TCP_DATA".MOD_DEVICE_STATION4[6].MASTER_READ_DATA.MOD_COIL_DATA[14] AND "S4_SENSOR_CYL6",   // "LPG_FILLING_FB"
                    INxAuto_Start_Seq := "MASTER_FILL_DATA".FILL_STATION_4[6].FILL_SEQ_IN.Auto_Start_Seq AND (12.0 < "hmi_dummy_array".S4_PrefillingDummyData[6].rTareWeight),
                    INxMan_Start_Seq := "MASTER_FILL_DATA".FILL_STATION_4[6].FILL_SEQ_IN.Man_Start_Seq,
                    INxStop_Sequence := "MASTER_FILL_DATA".FILL_STATION_4[6].FILL_SEQ_IN.Stop_Seq,
                    INtStart_TImeout_Time := "MASTER_FILL_DATA".FILL_STATION_4[6].FILL_SEQ_IN.Start_Timeout_Sec,
                    INxReset_Sequence := "MASTER_FILL_DATA".FILL_STATION_4[6].FILL_SEQ_IN.Reset_Seq,
                    INxCylinder_Type := "hmi_dummy_array".S4_PrefillingDummyData[6].iCylinderType,
                    INrTare_Entry_SP := "hmi_dummy_array".S4_PrefillingDummyData[6].rTareWeight,
                    ALL_FILL_DONE := "FILLING_STATION4_DB".FILLING_STATION4.ALL_FILL_DONE,
                    DOWN_CONVEYOR := "S4_DOWN_CONVEYOR",
                    Modbus_Master_DB := "MASTER_TCP_DATA".MOD_DEVICE_STATION4[6],
                    OutuFilled_Data => "MASTER_FILL_DATA".FILL_STATION_4[6].FILL_SEQ_OUT.Filled_Dat,
                    OutxDomestic_Cylinder => "MASTER_FILL_DATA".FILL_STATION_4[6].FILL_SEQ_OUT.Domestic_Cyl,
                    OutxCommercial_Cylinder => "MASTER_FILL_DATA".FILL_STATION_4[6].FILL_SEQ_OUT.Commercial_Cyl,
                    OutxStart_Timeout => %DB504.DBX27.0,
                    OutxTare_Entry_Error => %DB504.DBX27.1,
                    Outx_Filling_Error => %DB504.DBX27.2,
                    Outx_Tare_Value_Error => %DB504.DBX27.3,
                    Cycle_Started => #FILL_SEQ_STARTED[6],
                    OutiStep_No => "MASTER_FILL_DATA".FILL_STATION_4[6].FILL_SEQ_OUT.Step_No,
                    OUTxFilling_Done => #FILLING_DONE[6],
                    Gross_Weight => "CylinderSetup_DB".Array_S6[6].rGross_Weight,
                    Net_Wieght => "CylinderSetup_DB".Array_S6[6].rNet_weight);
   END_IF;
END_REGION

REGION Network 9: Reset Sequence
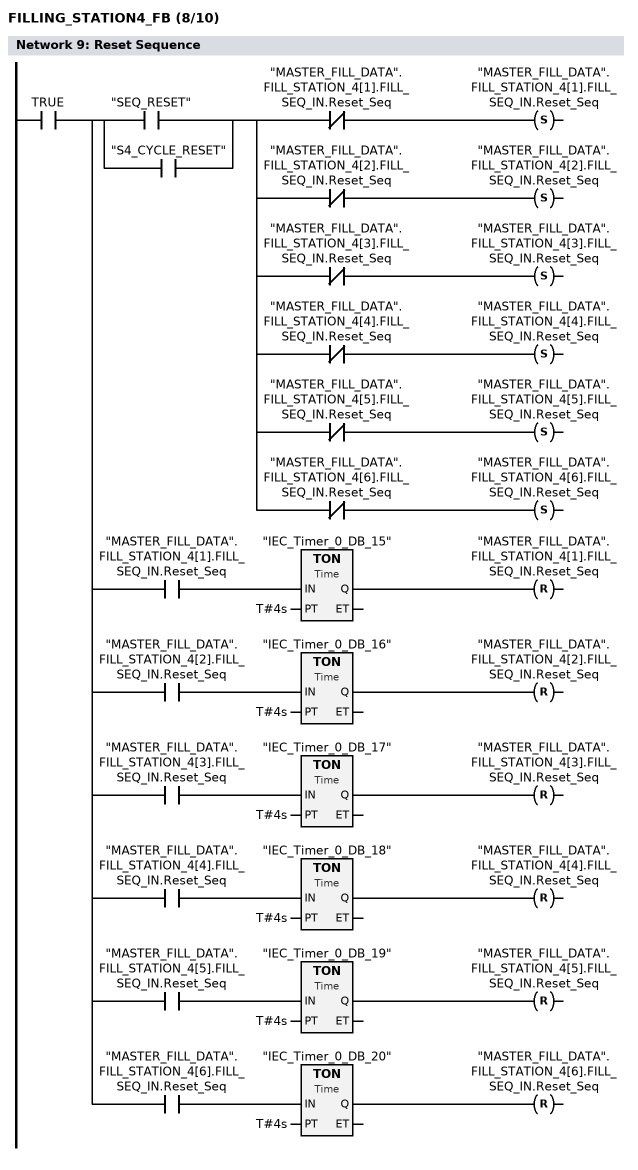
   RUNG wire#powerrail
      Contact( TRUE )
      wire#w1
      Contact( "SEQ_RESET" )
      wire#w2
      I_Contact( "MASTER_FILL_DATA".FILL_STATION_4[1].FILL_SEQ_IN.Reset_Seq )
      S_Coil( "MASTER_FILL_DATA".FILL_STATION_4[1].FILL_SEQ_IN.Reset_Seq )
   END_RUNG
   RUNG wire#w1
      Contact( "S4_CYCLE_RESET" )
   END_RUNG wire#w2
   RUNG wire#w2
      I_Contact( "MASTER_FILL_DATA".FILL_STATION_4[2].FILL_SEQ_IN.Reset_Seq )
      S_Coil( "MASTER_FILL_DATA".FILL_STATION_4[2].FILL_SEQ_IN.Reset_Seq )
   END_RUNG
   RUNG wire#w2
      I_Contact( "MASTER_FILL_DATA".FILL_STATION_4[3].FILL_SEQ_IN.Reset_Seq )
      S_Coil( "MASTER_FILL_DATA".FILL_STATION_4[3].FILL_SEQ_IN.Reset_Seq )
   END_RUNG
   RUNG wire#w2
      I_Contact( "MASTER_FILL_DATA".FILL_STATION_4[4].FILL_SEQ_IN.Reset_Seq )
      S_Coil( "MASTER_FILL_DATA".FILL_STATION_4[4].FILL_SEQ_IN.Reset_Seq )
   END_RUNG
   RUNG wire#w2
      I_Contact( "MASTER_FILL_DATA".FILL_STATION_4[5].FILL_SEQ_IN.Reset_Seq )
      S_Coil( "MASTER_FILL_DATA".FILL_STATION_4[5].FILL_SEQ_IN.Reset_Seq )
   END_RUNG
   RUNG wire#w2
      I_Contact( "MASTER_FILL_DATA".FILL_STATION_4[6].FILL_SEQ_IN.Reset_Seq )
      S_Coil( "MASTER_FILL_DATA".FILL_STATION_4[6].FILL_SEQ_IN.Reset_Seq )
   END_RUNG
   RUNG wire#w1
      Contact( "MASTER_FILL_DATA".FILL_STATION_4[1].FILL_SEQ_IN.Reset_Seq )
      { S7_Templates := "time_type := Time" } "IEC_Timer_0_DB_15".TON(pt := T#4s, et =>)
      R_Coil( "MASTER_FILL_DATA".FILL_STATION_4[1].FILL_SEQ_IN.Reset_Seq )
   END_RUNG
   RUNG wire#w1
      Contact( "MASTER_FILL_DATA".FILL_STATION_4[2].FILL_SEQ_IN.Reset_Seq )
      { S7_Templates := "time_type := Time" } "IEC_Timer_0_DB_16".TON(pt := T#4s, et =>)
      R_Coil( "MASTER_FILL_DATA".FILL_STATION_4[2].FILL_SEQ_IN.Reset_Seq )
   END_RUNG
   RUNG wire#w1
      Contact( "MASTER_FILL_DATA".FILL_STATION_4[3].FILL_SEQ_IN.Reset_Seq )
      { S7_Templates := "time_type := Time" } "IEC_Timer_0_DB_17".TON(pt := T#4s, et =>)
      R_Coil( "MASTER_FILL_DATA".FILL_STATION_4[3].FILL_SEQ_IN.Reset_Seq )
   END_RUNG
   RUNG wire#w1
      Contact( "MASTER_FILL_DATA".FILL_STATION_4[4].FILL_SEQ_IN.Reset_Seq )
      { S7_Templates := "time_type := Time" } "IEC_Timer_0_DB_18".TON(pt := T#4s, et =>)
      R_Coil( "MASTER_FILL_DATA".FILL_STATION_4[4].FILL_SEQ_IN.Reset_Seq )
   END_RUNG
   RUNG wire#w1
      Contact( "MASTER_FILL_DATA".FILL_STATION_4[5].FILL_SEQ_IN.Reset_Seq )
      { S7_Templates := "time_type := Time" } "IEC_Timer_0_DB_19".TON(pt := T#4s, et =>)
      R_Coil( "MASTER_FILL_DATA".FILL_STATION_4[5].FILL_SEQ_IN.Reset_Seq )
   END_RUNG
   RUNG wire#w1
      Contact( "MASTER_FILL_DATA".FILL_STATION_4[6].FILL_SEQ_IN.Reset_Seq )
      { S7_Templates := "time_type := Time" } "IEC_Timer_0_DB_20".TON(pt := T#4s, et =>)
      R_Coil( "MASTER_FILL_DATA".FILL_STATION_4[6].FILL_SEQ_IN.Reset_Seq )
   END_RUNG
   // the same network as SCL:
   #_w1 := TRUE AND ("SEQ_RESET" OR "S4_CYCLE_RESET");
   IF #_w1 AND NOT "MASTER_FILL_DATA".FILL_STATION_4[1].FILL_SEQ_IN.Reset_Seq THEN
       "MASTER_FILL_DATA".FILL_STATION_4[1].FILL_SEQ_IN.Reset_Seq := TRUE;
   END_IF;
   IF #_w1 AND NOT "MASTER_FILL_DATA".FILL_STATION_4[2].FILL_SEQ_IN.Reset_Seq THEN
       "MASTER_FILL_DATA".FILL_STATION_4[2].FILL_SEQ_IN.Reset_Seq := TRUE;
   END_IF;
   IF #_w1 AND NOT "MASTER_FILL_DATA".FILL_STATION_4[3].FILL_SEQ_IN.Reset_Seq THEN
       "MASTER_FILL_DATA".FILL_STATION_4[3].FILL_SEQ_IN.Reset_Seq := TRUE;
   END_IF;
   IF #_w1 AND NOT "MASTER_FILL_DATA".FILL_STATION_4[4].FILL_SEQ_IN.Reset_Seq THEN
       "MASTER_FILL_DATA".FILL_STATION_4[4].FILL_SEQ_IN.Reset_Seq := TRUE;
   END_IF;
   IF #_w1 AND NOT "MASTER_FILL_DATA".FILL_STATION_4[5].FILL_SEQ_IN.Reset_Seq THEN
       "MASTER_FILL_DATA".FILL_STATION_4[5].FILL_SEQ_IN.Reset_Seq := TRUE;
   END_IF;
   IF #_w1 AND NOT "MASTER_FILL_DATA".FILL_STATION_4[6].FILL_SEQ_IN.Reset_Seq THEN
       "MASTER_FILL_DATA".FILL_STATION_4[6].FILL_SEQ_IN.Reset_Seq := TRUE;
   END_IF;
   "IEC_Timer_0_DB_15".TON(IN := TRUE AND "MASTER_FILL_DATA".FILL_STATION_4[1].FILL_SEQ_IN.Reset_Seq,
                           PT := T#4s);
   IF "IEC_Timer_0_DB_15".Q THEN "MASTER_FILL_DATA".FILL_STATION_4[1].FILL_SEQ_IN.Reset_Seq := FALSE; END_IF;
   "IEC_Timer_0_DB_16".TON(IN := TRUE AND "MASTER_FILL_DATA".FILL_STATION_4[2].FILL_SEQ_IN.Reset_Seq,
                           PT := T#4s);
   IF "IEC_Timer_0_DB_16".Q THEN "MASTER_FILL_DATA".FILL_STATION_4[2].FILL_SEQ_IN.Reset_Seq := FALSE; END_IF;
   "IEC_Timer_0_DB_17".TON(IN := TRUE AND "MASTER_FILL_DATA".FILL_STATION_4[3].FILL_SEQ_IN.Reset_Seq,
                           PT := T#4s);
   IF "IEC_Timer_0_DB_17".Q THEN "MASTER_FILL_DATA".FILL_STATION_4[3].FILL_SEQ_IN.Reset_Seq := FALSE; END_IF;
   "IEC_Timer_0_DB_18".TON(IN := TRUE AND "MASTER_FILL_DATA".FILL_STATION_4[4].FILL_SEQ_IN.Reset_Seq,
                           PT := T#4s);
   IF "IEC_Timer_0_DB_18".Q THEN "MASTER_FILL_DATA".FILL_STATION_4[4].FILL_SEQ_IN.Reset_Seq := FALSE; END_IF;
   "IEC_Timer_0_DB_19".TON(IN := TRUE AND "MASTER_FILL_DATA".FILL_STATION_4[5].FILL_SEQ_IN.Reset_Seq,
                           PT := T#4s);
   IF "IEC_Timer_0_DB_19".Q THEN "MASTER_FILL_DATA".FILL_STATION_4[5].FILL_SEQ_IN.Reset_Seq := FALSE; END_IF;
   "IEC_Timer_0_DB_20".TON(IN := TRUE AND "MASTER_FILL_DATA".FILL_STATION_4[6].FILL_SEQ_IN.Reset_Seq,
                           PT := T#4s);
   IF "IEC_Timer_0_DB_20".Q THEN "MASTER_FILL_DATA".FILL_STATION_4[6].FILL_SEQ_IN.Reset_Seq := FALSE; END_IF;
END_REGION

REGION Network 10: Reset Sequence
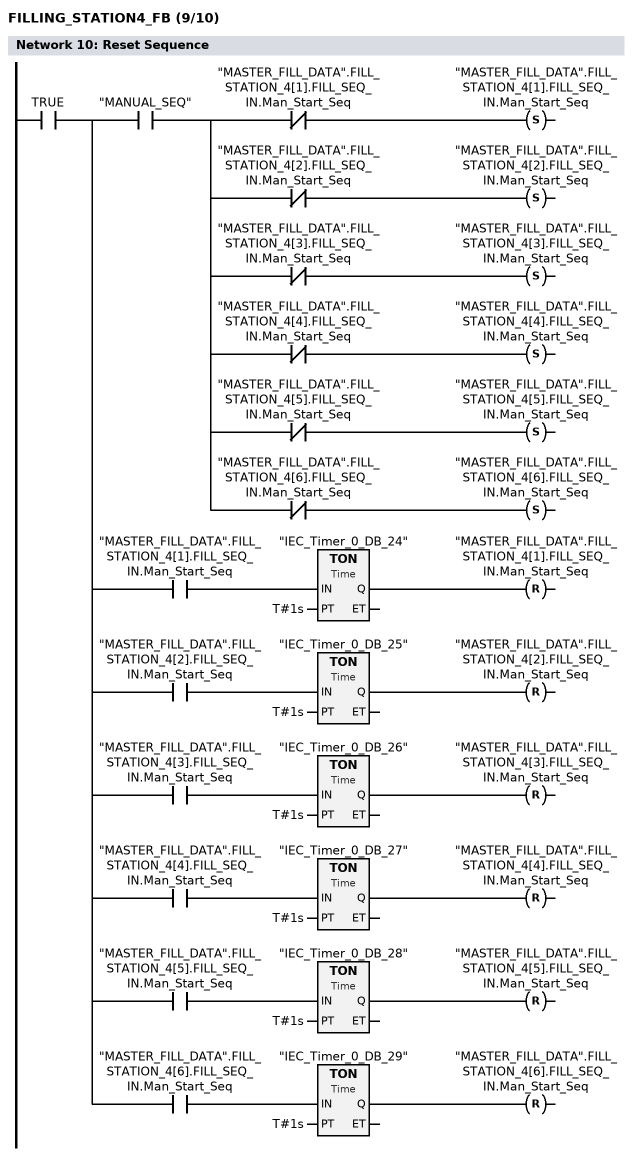
   RUNG wire#powerrail
      Contact( TRUE )
      wire#w1
      Contact( "MANUAL_SEQ" )
      wire#w2
      I_Contact( "MASTER_FILL_DATA".FILL_STATION_4[1].FILL_SEQ_IN.Man_Start_Seq )
      S_Coil( "MASTER_FILL_DATA".FILL_STATION_4[1].FILL_SEQ_IN.Man_Start_Seq )
   END_RUNG
   RUNG wire#w2
      I_Contact( "MASTER_FILL_DATA".FILL_STATION_4[2].FILL_SEQ_IN.Man_Start_Seq )
      S_Coil( "MASTER_FILL_DATA".FILL_STATION_4[2].FILL_SEQ_IN.Man_Start_Seq )
   END_RUNG
   RUNG wire#w2
      I_Contact( "MASTER_FILL_DATA".FILL_STATION_4[3].FILL_SEQ_IN.Man_Start_Seq )
      S_Coil( "MASTER_FILL_DATA".FILL_STATION_4[3].FILL_SEQ_IN.Man_Start_Seq )
   END_RUNG
   RUNG wire#w2
      I_Contact( "MASTER_FILL_DATA".FILL_STATION_4[4].FILL_SEQ_IN.Man_Start_Seq )
      S_Coil( "MASTER_FILL_DATA".FILL_STATION_4[4].FILL_SEQ_IN.Man_Start_Seq )
   END_RUNG
   RUNG wire#w2
      I_Contact( "MASTER_FILL_DATA".FILL_STATION_4[5].FILL_SEQ_IN.Man_Start_Seq )
      S_Coil( "MASTER_FILL_DATA".FILL_STATION_4[5].FILL_SEQ_IN.Man_Start_Seq )
   END_RUNG
   RUNG wire#w2
      I_Contact( "MASTER_FILL_DATA".FILL_STATION_4[6].FILL_SEQ_IN.Man_Start_Seq )
      S_Coil( "MASTER_FILL_DATA".FILL_STATION_4[6].FILL_SEQ_IN.Man_Start_Seq )
   END_RUNG
   RUNG wire#w1
      Contact( "MASTER_FILL_DATA".FILL_STATION_4[1].FILL_SEQ_IN.Man_Start_Seq )
      { S7_Templates := "time_type := Time" } "IEC_Timer_0_DB_24".TON(pt := T#1s, et =>)
      R_Coil( "MASTER_FILL_DATA".FILL_STATION_4[1].FILL_SEQ_IN.Man_Start_Seq )
   END_RUNG
   RUNG wire#w1
      Contact( "MASTER_FILL_DATA".FILL_STATION_4[2].FILL_SEQ_IN.Man_Start_Seq )
      { S7_Templates := "time_type := Time" } "IEC_Timer_0_DB_25".TON(pt := T#1s, et =>)
      R_Coil( "MASTER_FILL_DATA".FILL_STATION_4[2].FILL_SEQ_IN.Man_Start_Seq )
   END_RUNG
   RUNG wire#w1
      Contact( "MASTER_FILL_DATA".FILL_STATION_4[3].FILL_SEQ_IN.Man_Start_Seq )
      { S7_Templates := "time_type := Time" } "IEC_Timer_0_DB_26".TON(pt := T#1s, et =>)
      R_Coil( "MASTER_FILL_DATA".FILL_STATION_4[3].FILL_SEQ_IN.Man_Start_Seq )
   END_RUNG
   RUNG wire#w1
      Contact( "MASTER_FILL_DATA".FILL_STATION_4[4].FILL_SEQ_IN.Man_Start_Seq )
      { S7_Templates := "time_type := Time" } "IEC_Timer_0_DB_27".TON(pt := T#1s, et =>)
      R_Coil( "MASTER_FILL_DATA".FILL_STATION_4[4].FILL_SEQ_IN.Man_Start_Seq )
   END_RUNG
   RUNG wire#w1
      Contact( "MASTER_FILL_DATA".FILL_STATION_4[5].FILL_SEQ_IN.Man_Start_Seq )
      { S7_Templates := "time_type := Time" } "IEC_Timer_0_DB_28".TON(pt := T#1s, et =>)
      R_Coil( "MASTER_FILL_DATA".FILL_STATION_4[5].FILL_SEQ_IN.Man_Start_Seq )
   END_RUNG
   RUNG wire#w1
      Contact( "MASTER_FILL_DATA".FILL_STATION_4[6].FILL_SEQ_IN.Man_Start_Seq )
      { S7_Templates := "time_type := Time" } "IEC_Timer_0_DB_29".TON(pt := T#1s, et =>)
      R_Coil( "MASTER_FILL_DATA".FILL_STATION_4[6].FILL_SEQ_IN.Man_Start_Seq )
   END_RUNG
   // the same network as SCL:
   #_w1 := TRUE AND "MANUAL_SEQ";
   IF #_w1 AND NOT "MASTER_FILL_DATA".FILL_STATION_4[1].FILL_SEQ_IN.Man_Start_Seq THEN
       "MASTER_FILL_DATA".FILL_STATION_4[1].FILL_SEQ_IN.Man_Start_Seq := TRUE;
   END_IF;
   IF #_w1 AND NOT "MASTER_FILL_DATA".FILL_STATION_4[2].FILL_SEQ_IN.Man_Start_Seq THEN
       "MASTER_FILL_DATA".FILL_STATION_4[2].FILL_SEQ_IN.Man_Start_Seq := TRUE;
   END_IF;
   IF #_w1 AND NOT "MASTER_FILL_DATA".FILL_STATION_4[3].FILL_SEQ_IN.Man_Start_Seq THEN
       "MASTER_FILL_DATA".FILL_STATION_4[3].FILL_SEQ_IN.Man_Start_Seq := TRUE;
   END_IF;
   IF #_w1 AND NOT "MASTER_FILL_DATA".FILL_STATION_4[4].FILL_SEQ_IN.Man_Start_Seq THEN
       "MASTER_FILL_DATA".FILL_STATION_4[4].FILL_SEQ_IN.Man_Start_Seq := TRUE;
   END_IF;
   IF #_w1 AND NOT "MASTER_FILL_DATA".FILL_STATION_4[5].FILL_SEQ_IN.Man_Start_Seq THEN
       "MASTER_FILL_DATA".FILL_STATION_4[5].FILL_SEQ_IN.Man_Start_Seq := TRUE;
   END_IF;
   IF #_w1 AND NOT "MASTER_FILL_DATA".FILL_STATION_4[6].FILL_SEQ_IN.Man_Start_Seq THEN
       "MASTER_FILL_DATA".FILL_STATION_4[6].FILL_SEQ_IN.Man_Start_Seq := TRUE;
   END_IF;
   "IEC_Timer_0_DB_24".TON(IN := TRUE AND "MASTER_FILL_DATA".FILL_STATION_4[1].FILL_SEQ_IN.Man_Start_Seq,
                           PT := T#1s);
   IF "IEC_Timer_0_DB_24".Q THEN
       "MASTER_FILL_DATA".FILL_STATION_4[1].FILL_SEQ_IN.Man_Start_Seq := FALSE;
   END_IF;
   "IEC_Timer_0_DB_25".TON(IN := TRUE AND "MASTER_FILL_DATA".FILL_STATION_4[2].FILL_SEQ_IN.Man_Start_Seq,
                           PT := T#1s);
   IF "IEC_Timer_0_DB_25".Q THEN
       "MASTER_FILL_DATA".FILL_STATION_4[2].FILL_SEQ_IN.Man_Start_Seq := FALSE;
   END_IF;
   "IEC_Timer_0_DB_26".TON(IN := TRUE AND "MASTER_FILL_DATA".FILL_STATION_4[3].FILL_SEQ_IN.Man_Start_Seq,
                           PT := T#1s);
   IF "IEC_Timer_0_DB_26".Q THEN
       "MASTER_FILL_DATA".FILL_STATION_4[3].FILL_SEQ_IN.Man_Start_Seq := FALSE;
   END_IF;
   "IEC_Timer_0_DB_27".TON(IN := TRUE AND "MASTER_FILL_DATA".FILL_STATION_4[4].FILL_SEQ_IN.Man_Start_Seq,
                           PT := T#1s);
   IF "IEC_Timer_0_DB_27".Q THEN
       "MASTER_FILL_DATA".FILL_STATION_4[4].FILL_SEQ_IN.Man_Start_Seq := FALSE;
   END_IF;
   "IEC_Timer_0_DB_28".TON(IN := TRUE AND "MASTER_FILL_DATA".FILL_STATION_4[5].FILL_SEQ_IN.Man_Start_Seq,
                           PT := T#1s);
   IF "IEC_Timer_0_DB_28".Q THEN
       "MASTER_FILL_DATA".FILL_STATION_4[5].FILL_SEQ_IN.Man_Start_Seq := FALSE;
   END_IF;
   "IEC_Timer_0_DB_29".TON(IN := TRUE AND "MASTER_FILL_DATA".FILL_STATION_4[6].FILL_SEQ_IN.Man_Start_Seq,
                           PT := T#1s);
   IF "IEC_Timer_0_DB_29".Q THEN
       "MASTER_FILL_DATA".FILL_STATION_4[6].FILL_SEQ_IN.Man_Start_Seq := FALSE;
   END_IF;
END_REGION

REGION Network 11
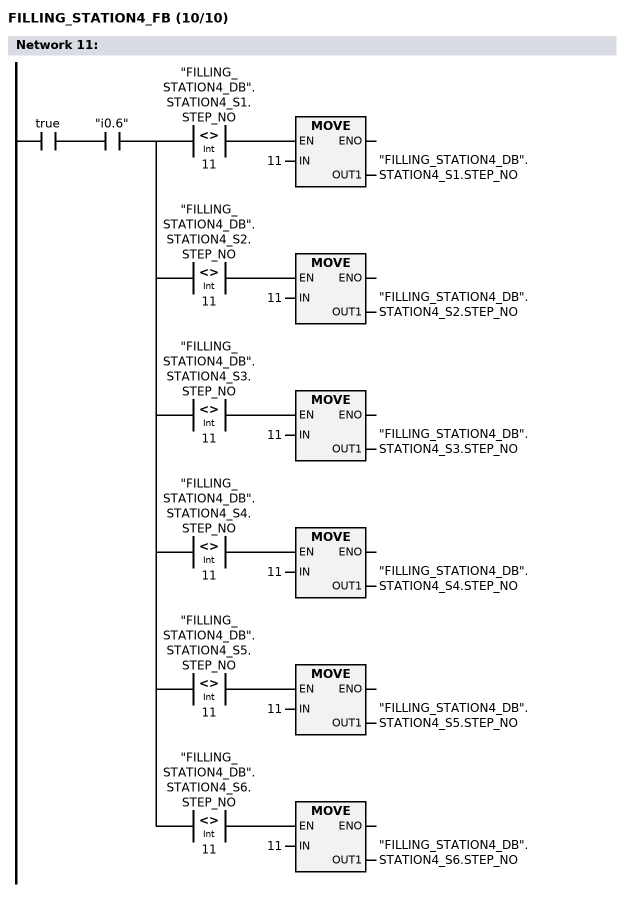
   RUNG wire#powerrail
      Contact( true )
      Contact( "i0.6" )
      wire#w1
      { S7_Templates := "SrcType := Int" } NE_Contact(in1 := "FILLING_STATION4_DB".STATION4_S1.STEP_NO, in2 := 11)
      Move(in := 11, out1 => "FILLING_STATION4_DB".STATION4_S1.STEP_NO)
   END_RUNG
   RUNG wire#w1
      { S7_Templates := "SrcType := Int" } NE_Contact(in1 := "FILLING_STATION4_DB".STATION4_S2.STEP_NO, in2 := 11)
      Move(in := 11, out1 => "FILLING_STATION4_DB".STATION4_S2.STEP_NO)
   END_RUNG
   RUNG wire#w1
      { S7_Templates := "SrcType := Int" } NE_Contact(in1 := "FILLING_STATION4_DB".STATION4_S3.STEP_NO, in2 := 11)
      Move(in := 11, out1 => "FILLING_STATION4_DB".STATION4_S3.STEP_NO)
   END_RUNG
   RUNG wire#w1
      { S7_Templates := "SrcType := Int" } NE_Contact(in1 := "FILLING_STATION4_DB".STATION4_S4.STEP_NO, in2 := 11)
      Move(in := 11, out1 => "FILLING_STATION4_DB".STATION4_S4.STEP_NO)
   END_RUNG
   RUNG wire#w1
      { S7_Templates := "SrcType := Int" } NE_Contact(in1 := "FILLING_STATION4_DB".STATION4_S5.STEP_NO, in2 := 11)
      Move(in := 11, out1 => "FILLING_STATION4_DB".STATION4_S5.STEP_NO)
   END_RUNG
   RUNG wire#w1
      { S7_Templates := "SrcType := Int" } NE_Contact(in1 := "FILLING_STATION4_DB".STATION4_S6.STEP_NO, in2 := 11)
      Move(in := 11, out1 => "FILLING_STATION4_DB".STATION4_S6.STEP_NO)
   END_RUNG
   // the same network as SCL:
   #_w1 := true AND "i0.6";
   IF #_w1 AND ("FILLING_STATION4_DB".STATION4_S1.STEP_NO <> 11) THEN
       "FILLING_STATION4_DB".STATION4_S1.STEP_NO := 11;
   END_IF;
   IF #_w1 AND ("FILLING_STATION4_DB".STATION4_S2.STEP_NO <> 11) THEN
       "FILLING_STATION4_DB".STATION4_S2.STEP_NO := 11;
   END_IF;
   IF #_w1 AND ("FILLING_STATION4_DB".STATION4_S3.STEP_NO <> 11) THEN
       "FILLING_STATION4_DB".STATION4_S3.STEP_NO := 11;
   END_IF;
   IF #_w1 AND ("FILLING_STATION4_DB".STATION4_S4.STEP_NO <> 11) THEN
       "FILLING_STATION4_DB".STATION4_S4.STEP_NO := 11;
   END_IF;
   IF #_w1 AND ("FILLING_STATION4_DB".STATION4_S5.STEP_NO <> 11) THEN
       "FILLING_STATION4_DB".STATION4_S5.STEP_NO := 11;
   END_IF;
   IF #_w1 AND ("FILLING_STATION4_DB".STATION4_S6.STEP_NO <> 11) THEN
       "FILLING_STATION4_DB".STATION4_S6.STEP_NO := 11;
   END_IF;
END_REGION
END_FUNCTION_BLOCK
